{attribute 'qualified_only'}
{attribute 'strict'}
TYPE E_MbOp :
(
	Read := 0,
	Write
);
END_TYPE

(* stored: Version 1.1.0.1
   DUT E_MbOp: Id {800f8a0d-d3f1-4d1e-a73e-c29985a03eda} *)
